// TIA Portal V17 export
// export: Created 2021-12-03T08:13:11.0357607Z, ExportSetting WithDefaults, DisplayName Totally Integrated Automation Portal, DisplayVersion V17, DisplayName TIA Portal Openness, DisplayVersion V17, DisplayName TIA Portal Version Control Interface, DisplayVersion V17, DisplayName STEP 7 Professional, DisplayVersion V17, DisplayName STEP 7 Safety, DisplayVersion V17, DisplayName WinCC Advanced, DisplayVersion V17
DATA_BLOCK "FGDB_EmStpButton"   // DB200, F_DB
VERSION : 0.1
// stored: AutoNumber false
   VAR
      P1EmStp_Sv : Bool;
      P1EmStp_Ev : Bool;
      P1EmStp_AckReq : Bool;
      P2EmStp_Sv : Bool;
      P2EmStp_Ev : Bool;
      P2EmStp_AckReq : Bool;
      P3EmStp_Sv : Bool;
      P3EmStp_Ev : Bool;
      P3EmStp_AckReq : Bool;
      AccEmStp_Sv : Bool;
      AccEmStp_Ev : Bool;
      AccEmStp_AckReq : Bool;
      DosimEmStp_Sv : Bool;
      DosimEmStp_Ev : Bool;
      DosimEmStp_AckReq : Bool;
      GnEmStp_Sv : Bool;
      GnEmStp_Ev : Bool;
      GnEmStp_AckReq : Bool;
   END_VAR
BEGIN
END_DATA_BLOCK
